TYPE CM_Sensor_CS :
STRUCT
	Auto		: BOOL;
	Manueel		: BOOL;
	Output		: BOOL;
END_STRUCT
END_TYPE

(* stored: Version 1.1.0.1, ProductVersion 3.1.4024.12
   DUT CM_Sensor_CS: Id {1d0887d0-2d70-4da0-8ef5-c7ef4e836e17} *)
